// TwinCAT 3 PLC project PLC
// ProgramVersion: 3.1.4024.0
// libraries:
//   EfficientIO Communicator, * (EfficientIO)
//   EfficientIO ModbusTCP, * (EfficientIO)
//   Lynus Energy Basic, * (Lynus AG)
//   Lynus Persistent Data V1, * (Lynus AG)
//   Lynus Standards, * (Lynus AG)
//   Tc2_Standard, * (Beckhoff Automation GmbH)
//   Tc2_System, * (Beckhoff Automation GmbH)
//   Tc3_Module, * (Beckhoff Automation GmbH)
// project tree:
//   / FastTast.TcTTO, MiddleTast.TcTTO, SlowTast.TcTTO
//   POUs/ prgCom.TcPOU, prgCS1.TcPOU, prgCS4.TcPOU, prgCS2.TcPOU, prgCS3.TcPOU, prgEM.TcPOU, prgEMS.TcPOU, prgGrid.TcPOU, prgPD.TcPOU (not stored), prgVar.TcPOU
// real-time tasks:
//   TASK FastTast: cycle T#5ms, priority 19, ADS port 351
//   TASK MiddleTast: cycle T#10ms, priority 20, ADS port 352
//   TASK SlowTast: cycle T#20ms, priority 21, ADS port 353

CONFIGURATION PLC
    RESOURCE PLC ON TwinCAT3
        TASK FastTast(INTERVAL := T#5ms, PRIORITY := 19);
        TASK MiddleTast(INTERVAL := T#10ms, PRIORITY := 20);
        TASK SlowTast(INTERVAL := T#20ms, PRIORITY := 21);
        PROGRAM prgVar WITH FastTast : prgVar;
        PROGRAM prgPD WITH FastTast : prgPD;
        PROGRAM prgEM WITH MiddleTast : prgEM;
        PROGRAM prgGrid WITH MiddleTast : prgGrid;
        PROGRAM prgEMS WITH MiddleTast : prgEMS;
        PROGRAM prgCS1 WITH MiddleTast : prgCS1;
        PROGRAM prgCS2 WITH MiddleTast : prgCS2;
        PROGRAM prgCS3 WITH MiddleTast : prgCS3;
        PROGRAM prgCS4 WITH MiddleTast : prgCS4;
        PROGRAM prgCom WITH SlowTast : prgCom;
    END_RESOURCE
END_CONFIGURATION

// ---- POUs/prgVar.TcPOU
PROGRAM prgVar
VAR
	fbVar			: FB_VarInfo_V3;
	fbrw1			: FB_ReadWrite_V2;
END_VAR

fbVar(
	bReadInfo:= , 
	eTMCFile:= eSelectTMCFile.eDontUseTMCFile, 
	eSavePositionTMCFile:= eSavePositionOnPLC.ePostionC, 
	udiCounterFoundVariables=> , 
	bError=> , 
	bBusy=> , 
	byProgress=> , 
	udiErrorCodeOut=> , 
	eErrorVarInfo_Out=> , 
	sVarWithError=> );
fbVar();
fbVar();	

fbRW1(	eUploadType := eSelectDataUploadType.e_Change_Intervall5min,
		bBusy=> , 
		bError=> , 
		udiErrorCodeOut=> , 
		eErrorReadWrite_Out=> );

END_PROGRAM

// ---- POUs/prgEM.TcPOU
PROGRAM prgEM
VAR
	FB_Phoenix:FB_PhoenixContact_EM_EEM_EM375;
	
	lrPower_Grid_TotalkW			: LREAL;			//{#lynus.ag#()}
	lrPower_Grid_L1				: LREAL;			//{#lynus.ag#()}
	lrPower_Grid_L2				: LREAL;			//{#lynus.ag#()}
	lrPower_Grid_L3				: LREAL;			//{#lynus.ag#()}
	lrCurrent_Grid_L1			: LREAL;			//{#lynus.ag#()}
	lrCurrent_Grid_L2			: LREAL;			//{#lynus.ag#()}
	lrCurrent_Grid_L3			: LREAL;			//{#lynus.ag#()}
	lrVoltage_Grid_L1N			: LREAL;			//{#lynus.ag#()}
	lrVoltage_Grid_L2N			: LREAL;			//{#lynus.ag#()}
	lrVoltage_Grid_L3N			: LREAL;			//{#lynus.ag#()}
	

	flEMPowerTotal		: LREAL;
	bPullSuccessfull 	: BOOL;
	udintErrorID		: UDINT;


	uint_State								AT%I* 	: uint;
	lrPower_House_kW			: LREAL;			//{#lynus.ag#()}
		
END_VAR

VAR PERSISTENT
	bEnableEM			: 	BOOL;
END_VAR


lrPower_House_kW := LIMIT(0,- FB_Phoenix.stDataEMPower.lrPowerTotal - prgCS1.lrPower_Alfen_S1 - prgCS2.lrPower_Alfen_S1 - prgCS3.lrPower_Alfen_S1 - prgCS4.lrPowerDC1_S1 - prgCS4.lrPowerDC1_S2,100);


FB_Phoenix(
	bEnable:= TRUE, 
	byUnitID:= 255, 
	sIPAdress:= '192.168.1.11', 
	stDataEMPower=> , 
	stDataEMCounter=> , 
	stDataEMPowerRealTime=> , 
	stDataEMCounterRealTime=> , 
	diNrOfEM_OUT=> );

	
lrPower_Grid_TotalkW 	:= 	-FB_Phoenix.stDataEMPower.lrPowerTotal;
lrPower_Grid_L1		 	:= 	-FB_Phoenix.stDataEMPower.lrPowerL1;
lrPower_Grid_L2		 	:= 	-FB_Phoenix.stDataEMPower.lrPowerL2;
lrPower_Grid_L3		 	:= 	-FB_Phoenix.stDataEMPower.lrPowerL3;
lrCurrent_Grid_L1 		:= 	FB_Phoenix.stDataEMPower.lrCurrentL1;
lrCurrent_Grid_L2 		:= 	FB_Phoenix.stDataEMPower.lrCurrentL2;
lrCurrent_Grid_L3 		:= 	FB_Phoenix.stDataEMPower.lrCurrentL3;
lrVoltage_Grid_L1N		:= 	FB_Phoenix.stDataEMPower.lrVoltageL1N;
lrVoltage_Grid_L2N		:= 	FB_Phoenix.stDataEMPower.lrVoltageL2N;
lrVoltage_Grid_L3N		:= 	FB_Phoenix.stDataEMPower.lrVoltageL3N;

END_PROGRAM

// ---- POUs/prgCS1.TcPOU
(*
----------------------------------- Alpitronic -----------------------------------
This Program is used for setting up Alpitronic Hyperchargers
*)

PROGRAM prgCS1
VAR
	fbAlfen						: FB_ECS_Alfen_NG9xx_Platform;
	bSManualyOn_Alfen				: BOOL;												//{#lynus.ag#()}
	bEnabled_Alfen				: BOOL;												//{#lynus.ag#()}
	bySManualyTargetPower_Alfen	: BYTE;												//{#lynus.ag#()}
	bySMinPowerECS_Alfen			: BYTE;												//{#lynus.ag#()}
	byErrorWarning_Alfen			: BYTE;												//{#lynus.ag#()}
	lrPowerTotal_Alfen			: LREAL;											//{#lynus.ag#()}
	lrPower_Alfen_S1				: LREAL;											//{#lynus.ag#()}
	lrPower_Alfen_S2				: LREAL;											//{#lynus.ag#()}
	rChargingTimeInMin_Alfen_S1	: REAL;												//{#lynus.ag#()}
	rChargingTimeInMin_Alfen_S2	: REAL;												//{#lynus.ag#()}
	rTargetPower_Alfen			: REAL;												//{#lynus.ag#()}
	wState_Alfen_S1				: WORD;												//{#lynus.ag#()}
	wState_Alfen_S2				: WORD;												//{#lynus.ag#()}
	lrEnergySession_Alfen_S1		: LREAL;											//{#lynus.ag#()}
	lrEnergySession_Alfen_S2		: LREAL;											//{#lynus.ag#()}
	lrTotalEnergy_Alfen			: LREAL;											//{#lynus.ag#()}
	bCarConnected_Alfen			: BOOL;												//{#lynus.ag#()}
	real_Target_Temp: REAL;
	liLPActualSurplusOrConsumption: INT;
	lrActualSurplusOrConsumption: LREAL;
	lreal_CSConsumptionTest: LREAL;
END_VAR

VAR PERSISTENT
	//Alfen
	bEnable_Alfen					: BOOL;												//{#lynus.ag#()}
	bManualyOn_Alfen				: BOOL;												//{#lynus.ag#()}
	byMinPower_Alfen				: BYTE;												//{#lynus.ag#()}
	byManualyTargetPower_Alfen	: BYTE;												//{#lynus.ag#()}
	byPrio_Alfen					: BYTE;												//{#lynus.ag#()}
	bySOCEnable_Alfen				: BYTE;												//{#lynus.ag#()}
	bySOCDisable_Alfen			: BYTE;												//{#lynus.ag#()}
	rMaxPower_Alfen				: REAL;												//{#lynus.ag#()}
	
END_VAR

				
(*-----------------------------------------------------------------------Alfen------------------------------------------------------*)

//Manual Power
fbAlfen.stSetupECS.bManualyOn := bManualyOn_Alfen;
fbAlfen.stSetupECS.byManualyTargetPower := byManualyTargetPower_Alfen;
fbAlfen.stSetupECS.byPriority := byPrio_Alfen;
fbAlfen.stSetupECS.byEnableSOC := bySOCEnable_Alfen;
fbAlfen.stSetupECS.byDisableSOC := bySOCDisable_Alfen;
fbAlfen.stSetupECS.rMaxPower := rMaxPower_Alfen;
fbAlfen.stSetupECS.byCSMinPower := byMinPower_Alfen;	

fbAlfen(
	bEnable:= bEnable_Alfen, 
	bPowerDataInvers:= , 
	byElectricFuseLine:= 1, 
	byUnitID_Socket1:= 1, 
	byUnitID_Socket2:= 2, 
	byNumberOfSockets:= 2,		//1 or 2. Depends on whether it is a single or double charging station  (Default: Single)
	byNumberOfConnectionWire:= 1, //1 or 2.  Depends on whether the charging station is supplied via a supply line or
	diNrOfEMS_IN:= prgEMS.fbEMS.diNrOfEMS_OUT, 
	diNrOfEM_IN_CS:= , 
	sIPAdress:= '192.168.1.21', 
	stSetupECS:= , 
	stDataECS=> , 
	diNrOfECS_OUT=> , 
	lrTotalPowerECSRealTime=> );						

bSManualyOn_Alfen := fbAlfen.stDataECS.bSManualyOn;
bySManualyTargetPower_Alfen := fbAlfen.stDataECS.bySManualyTargetPower;
byErrorWarning_Alfen := fbAlfen.stDataECS.byErrorWarning;
lrPowerTotal_Alfen := fbAlfen.stDataECS.lrTotalPower;
lrPower_Alfen_S1 :=  fbAlfen.stDataECS.arrSocketPower[1];
lrPower_Alfen_S2 :=  fbAlfen.stDataECS.arrSocketPower[2];
rChargingTimeInMin_Alfen_S1 := fbAlfen.stDataECS.arrChargingTimeInMin[1];
rChargingTimeInMin_Alfen_S2 := fbAlfen.stDataECS.arrChargingTimeInMin[2];		
wState_Alfen_S1 := fbAlfen.stDataECS.arrSocketStateECS[1];
wState_Alfen_S2 := fbAlfen.stDataECS.arrSocketStateECS[2];
lrEnergySession_Alfen_S1 := fbAlfen.stDataECS.arrSocketEnergySession[1];
lrEnergySession_Alfen_S2 := fbAlfen.stDataECS.arrSocketEnergySession[2];
lrTotalEnergy_Alfen := fbAlfen.stDataECS.lrTotalCounterEnergy_Consumption;
bySMinPowerECS_Alfen := fbAlfen.stDataECS.bySCSMinPower;
rTargetPower_Alfen := fbAlfen.stDataECS.rTargetPower;
bEnabled_Alfen := fbAlfen.stDataECS.bEnabled;
bCarConnected_Alfen := fbAlfen.stDataECS.bCarConnected;

END_PROGRAM

// ---- POUs/prgEMS.TcPOU
PROGRAM prgEMS
VAR PERSISTENT
	byMaxDepthOfDischrgEPO		: BYTE;							//{#lynus.ag#()}
	byPrioMinChrgBattSOCInEPO	: BYTE;							//{#lynus.ag#()}
	byResChrgfromGridToBatt		: BYTE;							//{#lynus.ag#()}
	byReserveSOCEPO				: BYTE;							//{#lynus.ag#()}
	uiUpdateTime				: UINT;							//{#lynus.ag#()}
	bEnableEMS					: BOOL;							//{#lynus.ag#()}
	bEnableMainFuse				: BOOL;							//{#lynus.ag#()}
	bAllowChrgFromGrid			: BOOL;							//{#lynus.ag#()}
	rMainFuseCSEMS				: REAL;							//{#lynus.ag#()}
	iOperationModeEMS			: INT;							//{#lynus.ag#()}
END_VAR
VAR
	fbEMS						: FB_EMS_V2;
	bIsEnableEMS				: BOOL;							//{#lynus.ag#()}
	bStateAllowChrgFromGrid		: BOOL;							//{#lynus.ag#()}
	bHPActivate					: BOOL;							//{#lynus.ag#()}
	bControllingState			: BOOL;							//{#lynus.ag#()}
	bSEnableMainFuse			: BOOL;							//{#lynus.ag#()}
	iMessageEMS					: INT;							//{#lynus.ag#()}
	rHeartbeatEMS				: REAL;							//{#lynus.ag#()}
	rErrorWarningEMS			: REAL;							//{#lynus.ag#()}
	rReadyEMS					: REAL;							//{#lynus.ag#()}
	rNewBatteryPowerEMS			: REAL;							//{#lynus.ag#()}
END_VAR

fbEMS.stSetupEMS.bAllowChrgFromGrid := bAllowChrgFromGrid;
fbEMS.stSetupEMS.byMaxDepthOfDischrgEPO := byMaxDepthOfDischrgEPO;
fbEMS.stSetupEMS.byPrioChrgBattSOCInEPO := byPrioMinChrgBattSOCInEPO;
fbEMS.stSetupEMS.byResChrgGridToBatt := byResChrgfromGridToBatt;
fbEMS.stSetupEMS.byReserveSOCEPO := byReserveSOCEPO;
fbEMS.stSizeMainFuseCS.rElSizeLine1 := rMainFuseCSEMS;
fbEMS.stSetupEMS.uiUpdateTime := uiUpdateTime;
fbEMS.stSetupEMS.bEnableMainFuseFunc := bEnableMainFuse;

IF iOperationModeEMS = 0 THEN fbEMS.eOperationMode := E_OperatingMode_EMS.eAllOff;
ELSIF iOperationModeEMS = 1 THEN fbEMS.eOperationMode := E_OperatingMode_EMS.eSelfConsumption;	
ELSIF iOperationModeEMS = 2 THEN fbEMS.eOperationMode := E_OperatingMode_EMS.ePeakLoadCapping;
ELSIF iOperationModeEMS = 3 THEN fbEMS.eOperationMode := E_OperatingMode_EMS.eLoadManagement;			
END_IF

fbEMS(
	bEnable:= bEnableEMS, 
	tDelayPwrCorrectionECS:= T#2.5S, 
	stNrOfEM_IN_ECS:= , 
	stSizeMainFuseCS:= , 
	stSetupEMS:= , 
	eOperationMode:= , 
	eSpeedModeBackendController:= E_SpeedModeBackendController_EMS.eSlow, 
	eSpeedModeLocalController:= E_SpeedModeLocalController_EMS.eSlow,
	bActivateHP:= bHPActivate, 
	bControllingState:= FALSE, //bControllingState, 
	rHeartbeat:= rHeartbeatEMS, 
	rErrorWarning:= rErrorWarningEMS, 
	rEnergyOptReady:= rReadyEMS, 
	rNewBattPower:= rNewBatteryPowerEMS, 
	eMessageEMS=> iMessageEMS, 
	bStateEnable=> bIsEnableEMS, 
	bStateAllowChrgFromGrid=> bStateAllowChrgFromGrid, 
	bMissingPowerData=> , 
	bSurplusAvailable=> , 
	bSEnableMainFuseFunc=> bSEnableMainFuse, 
	byProgress=> , 
	uiState_OUT=> , 
	diNrOfEMS_OUT=> , 
	arrMinPrioReached=> , 
	arrMaxPrioReached=> );

END_PROGRAM

// ---- POUs/prgCS2.TcPOU
(*
----------------------------------- Alpitronic -----------------------------------
This Program is used for setting up Alpitronic Hyperchargers
*)

PROGRAM prgCS2
VAR
	fbAlfen						: FB_ECS_Alfen_NG9xx_Platform;
	bSManualyOn_Alfen				: BOOL;												//{#lynus.ag#()}
	bEnabled_Alfen				: BOOL;												//{#lynus.ag#()}
	bySManualyTargetPower_Alfen	: BYTE;												//{#lynus.ag#()}
	bySMinPowerECS_Alfen			: BYTE;												//{#lynus.ag#()}
	byErrorWarning_Alfen			: BYTE;												//{#lynus.ag#()}
	lrPowerTotal_Alfen			: LREAL;											//{#lynus.ag#()}
	lrPower_Alfen_S1				: LREAL;											//{#lynus.ag#()}
	lrPower_Alfen_S2				: LREAL;											//{#lynus.ag#()}
	rChargingTimeInMin_Alfen_S1	: REAL;												//{#lynus.ag#()}
	rChargingTimeInMin_Alfen_S2	: REAL;												//{#lynus.ag#()}
	rTargetPower_Alfen			: REAL;												//{#lynus.ag#()}
	wState_Alfen_S1				: WORD;												//{#lynus.ag#()}
	wState_Alfen_S2				: WORD;												//{#lynus.ag#()}
	lrEnergySession_Alfen_S1		: LREAL;											//{#lynus.ag#()}
	lrEnergySession_Alfen_S2		: LREAL;											//{#lynus.ag#()}
	lrTotalEnergy_Alfen			: LREAL;											//{#lynus.ag#()}
	bCarConnected_Alfen			: BOOL;												//{#lynus.ag#()}
	real_Target_Temp: REAL;
	liLPActualSurplusOrConsumption: INT;
	lrActualSurplusOrConsumption: LREAL;
	lreal_CSConsumptionTest: LREAL;
END_VAR

VAR PERSISTENT
	//Alfen
	bEnable_Alfen					: BOOL;												//{#lynus.ag#()}
	bManualyOn_Alfen				: BOOL;												//{#lynus.ag#()}
	byMinPower_Alfen				: BYTE;												//{#lynus.ag#()}
	byManualyTargetPower_Alfen	: BYTE;												//{#lynus.ag#()}
	byPrio_Alfen					: BYTE;												//{#lynus.ag#()}
	bySOCEnable_Alfen				: BYTE;												//{#lynus.ag#()}
	bySOCDisable_Alfen			: BYTE;												//{#lynus.ag#()}
	rMaxPower_Alfen				: REAL;												//{#lynus.ag#()}
	
END_VAR

				
(*-----------------------------------------------------------------------Alfen------------------------------------------------------*)

//Manual Power
fbAlfen.stSetupECS.bManualyOn := bManualyOn_Alfen;
fbAlfen.stSetupECS.byManualyTargetPower := byManualyTargetPower_Alfen;
fbAlfen.stSetupECS.byPriority := byPrio_Alfen;
fbAlfen.stSetupECS.byEnableSOC := bySOCEnable_Alfen;
fbAlfen.stSetupECS.byDisableSOC := bySOCDisable_Alfen;
fbAlfen.stSetupECS.rMaxPower := rMaxPower_Alfen;
fbAlfen.stSetupECS.byCSMinPower := byMinPower_Alfen;	

fbAlfen(
	bEnable:= bEnable_Alfen, 
	bPowerDataInvers:= , 
	byElectricFuseLine:= 1, 
	byUnitID_Socket1:= 1, 
	byUnitID_Socket2:= 2, 
	byNumberOfSockets:= 2,		//1 or 2. Depends on whether it is a single or double charging station  (Default: Single)
	byNumberOfConnectionWire:= 1, //1 or 2.  Depends on whether the charging station is supplied via a supply line or
	diNrOfEMS_IN:= prgEMS.fbEMS.diNrOfEMS_OUT, 
	diNrOfEM_IN_CS:= , 
	sIPAdress:= '192.168.1.22', 
	stSetupECS:= , 
	stDataECS=> , 
	diNrOfECS_OUT=> , 
	lrTotalPowerECSRealTime=> );						

bSManualyOn_Alfen := fbAlfen.stDataECS.bSManualyOn;
bySManualyTargetPower_Alfen := fbAlfen.stDataECS.bySManualyTargetPower;
byErrorWarning_Alfen := fbAlfen.stDataECS.byErrorWarning;
lrPowerTotal_Alfen := fbAlfen.stDataECS.lrTotalPower;
lrPower_Alfen_S1 :=  fbAlfen.stDataECS.arrSocketPower[1];
lrPower_Alfen_S2 :=  fbAlfen.stDataECS.arrSocketPower[2];
rChargingTimeInMin_Alfen_S1 := fbAlfen.stDataECS.arrChargingTimeInMin[1];
rChargingTimeInMin_Alfen_S2 := fbAlfen.stDataECS.arrChargingTimeInMin[2];		
wState_Alfen_S1 := fbAlfen.stDataECS.arrSocketStateECS[1];
wState_Alfen_S2 := fbAlfen.stDataECS.arrSocketStateECS[2];
lrEnergySession_Alfen_S1 := fbAlfen.stDataECS.arrSocketEnergySession[1];
lrEnergySession_Alfen_S2 := fbAlfen.stDataECS.arrSocketEnergySession[2];
lrTotalEnergy_Alfen := fbAlfen.stDataECS.lrTotalCounterEnergy_Consumption;
bySMinPowerECS_Alfen := fbAlfen.stDataECS.bySCSMinPower;
rTargetPower_Alfen := fbAlfen.stDataECS.rTargetPower;
bEnabled_Alfen := fbAlfen.stDataECS.bEnabled;
bCarConnected_Alfen := fbAlfen.stDataECS.bCarConnected;

END_PROGRAM

// ---- POUs/prgCS3.TcPOU
(*
----------------------------------- Alpitronic -----------------------------------
This Program is used for setting up Alpitronic Hyperchargers
*)

PROGRAM prgCS3
VAR
	fbAlfen						: FB_ECS_Alfen_NG9xx_Platform;
	bSManualyOn_Alfen				: BOOL;												//{#lynus.ag#()}
	bEnabled_Alfen				: BOOL;												//{#lynus.ag#()}
	bySManualyTargetPower_Alfen	: BYTE;												//{#lynus.ag#()}
	bySMinPowerECS_Alfen			: BYTE;												//{#lynus.ag#()}
	byErrorWarning_Alfen			: BYTE;												//{#lynus.ag#()}
	lrPowerTotal_Alfen			: LREAL;											//{#lynus.ag#()}
	lrPower_Alfen_S1				: LREAL;											//{#lynus.ag#()}
	lrPower_Alfen_S2				: LREAL;											//{#lynus.ag#()}
	rChargingTimeInMin_Alfen_S1	: REAL;												//{#lynus.ag#()}
	rChargingTimeInMin_Alfen_S2	: REAL;												//{#lynus.ag#()}
	rTargetPower_Alfen			: REAL;												//{#lynus.ag#()}
	wState_Alfen_S1				: WORD;												//{#lynus.ag#()}
	wState_Alfen_S2				: WORD;												//{#lynus.ag#()}
	lrEnergySession_Alfen_S1		: LREAL;											//{#lynus.ag#()}
	lrEnergySession_Alfen_S2		: LREAL;											//{#lynus.ag#()}
	lrTotalEnergy_Alfen			: LREAL;											//{#lynus.ag#()}
	bCarConnected_Alfen			: BOOL;												//{#lynus.ag#()}
	real_Target_Temp: REAL;
	liLPActualSurplusOrConsumption: INT;
	lrActualSurplusOrConsumption: LREAL;
	lreal_CSConsumptionTest: LREAL;
END_VAR

VAR PERSISTENT
	//Alfen
	bEnable_Alfen					: BOOL;												//{#lynus.ag#()}
	bManualyOn_Alfen				: BOOL;												//{#lynus.ag#()}
	byMinPower_Alfen				: BYTE;												//{#lynus.ag#()}
	byManualyTargetPower_Alfen	: BYTE;												//{#lynus.ag#()}
	byPrio_Alfen					: BYTE;												//{#lynus.ag#()}
	bySOCEnable_Alfen				: BYTE;												//{#lynus.ag#()}
	bySOCDisable_Alfen			: BYTE;												//{#lynus.ag#()}
	rMaxPower_Alfen				: REAL;												//{#lynus.ag#()}
	
END_VAR

				
(*-----------------------------------------------------------------------Alfen------------------------------------------------------*)

//Manual Power
fbAlfen.stSetupECS.bManualyOn := bManualyOn_Alfen;
fbAlfen.stSetupECS.byManualyTargetPower := byManualyTargetPower_Alfen;
fbAlfen.stSetupECS.byPriority := byPrio_Alfen;
fbAlfen.stSetupECS.byEnableSOC := bySOCEnable_Alfen;
fbAlfen.stSetupECS.byDisableSOC := bySOCDisable_Alfen;
fbAlfen.stSetupECS.rMaxPower := rMaxPower_Alfen;
fbAlfen.stSetupECS.byCSMinPower := byMinPower_Alfen;	

fbAlfen(
	bEnable:= bEnable_Alfen, 
	bPowerDataInvers:= , 
	byElectricFuseLine:= 1, 
	byUnitID_Socket1:= 1, 
	byUnitID_Socket2:= 2, 
	byNumberOfSockets:= 2,		//1 or 2. Depends on whether it is a single or double charging station  (Default: Single)
	byNumberOfConnectionWire:= 1, //1 or 2.  Depends on whether the charging station is supplied via a supply line or
	diNrOfEMS_IN:= prgEMS.fbEMS.diNrOfEMS_OUT, 
	diNrOfEM_IN_CS:= , 
	sIPAdress:= '192.168.1.23', 
	stSetupECS:= , 
	stDataECS=> , 
	diNrOfECS_OUT=> , 
	lrTotalPowerECSRealTime=> );						

bSManualyOn_Alfen := fbAlfen.stDataECS.bSManualyOn;
bySManualyTargetPower_Alfen := fbAlfen.stDataECS.bySManualyTargetPower;
byErrorWarning_Alfen := fbAlfen.stDataECS.byErrorWarning;
lrPowerTotal_Alfen := fbAlfen.stDataECS.lrTotalPower;
lrPower_Alfen_S1 :=  fbAlfen.stDataECS.arrSocketPower[1];
lrPower_Alfen_S2 :=  fbAlfen.stDataECS.arrSocketPower[2];
rChargingTimeInMin_Alfen_S1 := fbAlfen.stDataECS.arrChargingTimeInMin[1];
rChargingTimeInMin_Alfen_S2 := fbAlfen.stDataECS.arrChargingTimeInMin[2];		
wState_Alfen_S1 := fbAlfen.stDataECS.arrSocketStateECS[1];
wState_Alfen_S2 := fbAlfen.stDataECS.arrSocketStateECS[2];
lrEnergySession_Alfen_S1 := fbAlfen.stDataECS.arrSocketEnergySession[1];
lrEnergySession_Alfen_S2 := fbAlfen.stDataECS.arrSocketEnergySession[2];
lrTotalEnergy_Alfen := fbAlfen.stDataECS.lrTotalCounterEnergy_Consumption;
bySMinPowerECS_Alfen := fbAlfen.stDataECS.bySCSMinPower;
rTargetPower_Alfen := fbAlfen.stDataECS.rTargetPower;
bEnabled_Alfen := fbAlfen.stDataECS.bEnabled;
bCarConnected_Alfen := fbAlfen.stDataECS.bCarConnected;

END_PROGRAM

// ---- POUs/prgCS4.TcPOU
PROGRAM prgCS4
VAR
	fbApliT					: FB_ECS_Alpitronic_Hypercharger;
	
	bSManualyOn_DC			: BOOL;												//{#lynus.ag#()}
	bEnabled					: BOOL;												//{#lynus.ag#()}
	bySManualyTargetPowerDC	: BYTE;												//{#lynus.ag#()}
	bySMinPowerECSDC			: BYTE;												//{#lynus.ag#()}
	byErrorWarningDC			: BYTE;												//{#lynus.ag#()}
	lrPowerTotalDC1				: LREAL;											//{#lynus.ag#()}
	lrPowerDC1_S1				: LREAL;											//{#lynus.ag#()}
	lrPowerDC1_S2				: LREAL;											//{#lynus.ag#()}
	lrPowerDC1_S3				: LREAL;											//{#lynus.ag#()}
	rChargingTimeInMinDC1_S1	: REAL;												//{#lynus.ag#()}
	rChargingTimeInMinDC1_S2	: REAL;												//{#lynus.ag#()}
	rChargingTimeInMinDC1_S3	: REAL;												//{#lynus.ag#()}
	rTargetPowerDC1				: REAL;												//{#lynus.ag#()}
	dwSOCCarDC1_S1				: DWORD;											//{#lynus.ag#()}
	dwSOCCarDC1_S2				: DWORD;											//{#lynus.ag#()}
	wStateDC1_S1				: WORD;												//{#lynus.ag#()}
	wStateDC1_S2				: WORD;												//{#lynus.ag#()}
	wStateDC1_S3				: WORD;												//{#lynus.ag#()}
	lrEnergySessionDC1_S1		: LREAL;											//{#lynus.ag#()}
	lrEnergySessionDC1_S2		: LREAL;											//{#lynus.ag#()}
	lrEnergySessionDC1_S3		: LREAL;											//{#lynus.ag#()}
	lrTotalEnergyDC1			: LREAL;											//{#lynus.ag#()}
	bCarConnected_DC1			: BOOL;												//{#lynus.ag#()}
	
END_VAR
VAR PERSISTENT
	bEnableDC1					: BOOL;												//{#lynus.ag#()}
	bManualyOnDC				: BOOL;												//{#lynus.ag#()}
	byMinPowerDC1				: BYTE;												//{#lynus.ag#()}
	byManualyTargetPowerDC	: BYTE;												//{#lynus.ag#()}
	byPrioDC1					: BYTE;												//{#lynus.ag#()}
	bySOCEnableDC1				: BYTE;												//{#lynus.ag#()}
	bySOCDisableDC1				: BYTE;												//{#lynus.ag#()}
	rMaxPowerDC1				: REAL;												//{#lynus.ag#()}
END_VAR

//Manual Power
fbApliT.stSetupECS.bManualyOn := bManualyOnDC;
fbApliT.stSetupECS.byManualyTargetPower := byManualyTargetPowerDC;
fbApliT.stSetupECS.byPriority := byPrioDC1;
fbApliT.stSetupECS.byEnableSOC := bySOCEnableDC1;
fbApliT.stSetupECS.byDisableSOC := bySOCDisableDC1;
fbApliT.stSetupECS.rMaxPower := rMaxPowerDC1;
fbApliT.stSetupECS.byCSMinPower := byMinPowerDC1;	
	
fbApliT(
	bEnable:= bEnableDC1, 
	bPowerDataInvers:= , 
	byElectricFuseLine:= , 
	byUnitID:= 1, 
	diNrOfEMS_IN:= prgEMS.fbEMS.diNrOfEMS_OUT, 
	diNrOfEM_IN_CS:= , 
	sIPAdress:= '192.168.1.24', 
	stSetupECS:= , 
	stDataECS=> , 
	diNrOfECS_OUT=> );

bSManualyOn_DC := fbApliT.stDataECS.bSManualyOn;
bySManualyTargetPowerDC := fbApliT.stDataECS.bySManualyTargetPower;
byErrorWarningDC := fbApliT.stDataECS.byErrorWarning;
lrPowerTotalDC1 := fbApliT.stDataECS.lrTotalPower;
lrPowerDC1_S1 :=  fbApliT.stDataECS.arrSocketPower[1];
lrPowerDC1_S2 :=  fbApliT.stDataECS.arrSocketPower[2];
lrPowerDC1_S3 := fbApliT.stDataECS.arrSocketPower[3];	 	
rChargingTimeInMinDC1_S1 := fbApliT.stDataECS.arrChargingTimeInMin[1];	
rChargingTimeInMinDC1_S2 := fbApliT.stDataECS.arrChargingTimeInMin[2];
rChargingTimeInMinDC1_S3 := fbApliT.stDataECS.arrChargingTimeInMin[3];
dwSOCCarDC1_S1 := fbApliT.stDataECS.arrSocketSOCCar[1]; 
dwSOCCarDC1_S2 := fbApliT.stDataECS.arrSocketSOCCar[2]; 	
wStateDC1_S1 := fbApliT.stDataECS.arrSocketStateECS[1];
wStateDC1_S2 := fbApliT.stDataECS.arrSocketStateECS[2];
wStateDC1_S3 := fbApliT.stDataECS.arrSocketStateECS[3];
lrEnergySessionDC1_S1 := fbApliT.stDataECS.arrSocketEnergySession[1];
lrEnergySessionDC1_S2 := fbApliT.stDataECS.arrSocketEnergySession[2];
lrEnergySessionDC1_S3 := fbApliT.stDataECS.arrSocketEnergySession[3];
lrTotalEnergyDC1 := fbApliT.stDataECS.lrTotalCounterEnergy_Consumption;
bySMinPowerECSDC := fbApliT.stDataECS.bySCSMinPower;
rTargetPowerDC1 := fbApliT.stDataECS.rTargetPower;
bEnabled := fbApliT.stDataECS.bEnabled;

bCarConnected_DC1 := fbApliT.stDataECS.bCarConnected;

END_PROGRAM

// ---- POUs/prgGrid.TcPOU
PROGRAM prgGrid
VAR PERSISTENT
	rSizeGridConn				: REAL;									//{#lynus.ag#()}
END_VAR
VAR
	fbGrid						: FB_Grid_Power_Ext_Input;
	lrGridPower					: LREAL;								//{#lynus.ag#()}
	lrGridPower_Consumption		: LREAL;								//{#lynus.ag#()}
	lrGridPower_Production		: LREAL;								//{#lynus.ag#()}
END_VAR

// the grid gets caluclated: House power + PV Power


fbGrid(
	bEnable:= TRUE, 
	diNrOfEMS_IN:= prgEMS.fbEMS.diNrOfEMS_OUT, 
	rSizeGridConn:= rSizeGridConn, 
	bExtErrorGrid:= , 
	lrExtGridPower:= prgEM.lrPower_Grid_TotalkW,	
	lrExtTotalCounterEnergy_Consumption:= 0, 
	lrExtTotalCounterEnergy_Production:= 0, 
	lrExtCounterEnergyT1_Consumption:= 0, 
	lrExtCounterEnergyT2_Consumption:= 0, 
	lrExtCounterEnergyT1_Production:= 0, 
	lrExtCounterEnergyT2_Production:= 0, 
	stDataGrid=> , 
	diNrOfGrid_OUT=> );
	
lrGridPower := fbGrid.stDataGrid.lrPower;
IF lrGridPower >=0 THEN 
	lrGridPower_Consumption := lrGridPower;
	lrGridPower_Production := 0;
ELSE
	lrGridPower_Consumption := 0;
	lrGridPower_Production := -lrGridPower;
END_IF

END_PROGRAM

// ---- POUs/prgCom.TcPOU
PROGRAM prgCom
VAR
	fbCom			: FB_MqttCommunicator_V3;
END_VAR

fbCom(
	bConnect:= TRUE,
	strAuthKey:= 'TSG88376368072',
	sUserName:= 'ab6b7704-0b2c-4c94-8e47-13d25c5f2bfa', 
	sUserPassword:= '78b266a9-af78-4bf8-8bad-800f54d6b5e5', 
	eSavePositionCertificate:= eSavePositionOnPLC.ePostionC, 
	bConnected=> , 
	bError=> , 
	hrErrorCode=> , 
	eConnectionState=> , 
	eErrorMessage_Out=> );

END_PROGRAM
